(* PLC project timer_counter, plcc plcc tests 1 *)
(* stored: creationDateTime 2026-09-27T00:00:00 *)

PROGRAM Machine
  VAR
    Enable : BOOL;
    Done : BOOL;
    Lamp : BOOL;
    Elapsed : TIME;
    T1 : TON;
    CountEn : BOOL;
    Pulse : BOOL;
    Reset : BOOL;
    Enabled : BOOL;
    Reached : BOOL;
    Count : INT;
    C1 : CTU;
  END_VAR

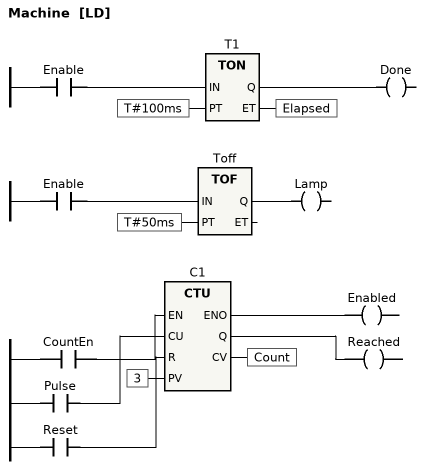
(* LD diagram, written out as Structured Text *)
T1(IN := Enable, PT := T#100ms);
Done := T1.Q;
Elapsed := T1.ET;
Toff(IN := Enable, PT := T#50ms);
Lamp := Toff.Q;
C1(EN := CountEn, CU := Pulse, R := Reset, PV := 3);
Enabled := C1.ENO;
Reached := C1.Q;
IF C1.ENO THEN Count := C1.CV; END_IF;
END_PROGRAM

CONFIGURATION Config0
  RESOURCE Res0 ON PLC
    TASK Cyclic(INTERVAL := T#10ms, PRIORITY := 0);
    PROGRAM machine WITH Cyclic : Machine;
  END_RESOURCE
END_CONFIGURATION
